TYPE (* The fixed type hash *)
  (* Standard: 61499-1; Description: Copyright (c) 2025 Martin Erich Jobst This program and the accompanying materials are made available under the terms of the Eclipse Public License 2.0 which is available at https://www.eclipse.org/legal/epl-2.0/ SPDX-License-Identifier: EPL-2.0 *)
  (* Version 1.0, 2025-06-05, Martin Erich Jobst, initial API and implementation and/or initial documentation *)
  PACKAGE eclipse4diac::core;
  {SET_ATTRIBUTE(TARGET, (IInterfaceElement:=FALSE,SubApp:=FALSE,FBType:=TRUE,Application:=FALSE,Connection:=FALSE,FB:=FALSE,DataType:=FALSE))}
  TypeHash : STRING := ''; (* The fixed type hash *)
END_TYPE
